// TwinCAT 3 PLC project MainProgram
// ProgramVersion: 3.1.4023.0
// libraries:
//   Tc2_Standard, * (Beckhoff Automation GmbH)
//   Tc2_System, * (Beckhoff Automation GmbH)
//   Tc3_Module, * (Beckhoff Automation GmbH)
// project tree:
//   DUT/ POS_Control.TcDUT, POS_Control_Control.TcDUT, POS_Status.TcDUT, POS_Status_Status.TcDUT, STM_Control.TcDUT, STM_Control_Control.TcDUT, STM_Status.TcDUT, STM_Status_Status.TcDUT, ST_PosInterface.TcDUT
//   GVLs/ GVL_IO.TcGVL
//   / PlcTask.TcTTO
//   POUs/ MAIN.TcPOU, POU_Example2PositionalMoves.TcPOU, POU_ExampleDynamicMoves.TcPOU
// real-time tasks:
//   TASK PlcTask: cycle T#10ms, priority 20, ADS port 350
//   TASK VnTask ImgAcq (FileSource1): cycle T#10ms, priority 5, ADS port 351
// I/O:
//   DEVICE Device 1 (Beckhoff CCAT)
//   DEVICE Device 2 (EtherCAT), AmsNetId 5.68.118.43.3.1
//     Term 1 (EK1200) [EK1200-5000 EtherCAT Power supply (2A E-Bus)]
//       Term 2 (EL7031) [EL7031 1Ch. Stepper motor output stage (24V, 1.5A)]
//       Term 3 (EL9011) [EL9011 End Terminal]
// variable links:
//   MainProgram Instance <-> Device 2 (EtherCAT)/Term 1 (EK1200)/Term 2 (EL7031)
//     PlcTask Inputs/GVL_IO.Axis.PosStatus/ActualDriveTime <-> POS Status/Actual drive time
//     PlcTask Inputs/GVL_IO.Axis.PosStatus/ActualPosition <-> POS Status/Actual position
//     PlcTask Inputs/GVL_IO.Axis.PosStatus/ActualVelocity <-> POS Status/Actual velocity
//     PlcTask Inputs/GVL_IO.Axis.PosStatus/Status <-> POS Status/Status
//     PlcTask Inputs/GVL_IO.Axis.StmStatus/Status <-> STM Status/Status
//     PlcTask Outputs/GVL_IO.Axis.PosControl/Acceleration <-> POS Control/Acceleration
//     PlcTask Outputs/GVL_IO.Axis.PosControl/Control <-> POS Control/Control
//     PlcTask Outputs/GVL_IO.Axis.PosControl/Deceleration <-> POS Control/Deceleration
//     PlcTask Outputs/GVL_IO.Axis.PosControl/StartType <-> POS Control/Start type
//     PlcTask Outputs/GVL_IO.Axis.PosControl/TargetPosition <-> POS Control/Target position
//     PlcTask Outputs/GVL_IO.Axis.PosControl/Velocity <-> POS Control/Velocity
//     PlcTask Outputs/GVL_IO.Axis.StmControl/Control <-> STM Control/Control

CONFIGURATION MainProgram
    RESOURCE PLC ON TwinCAT3
        TASK PlcTask(INTERVAL := T#10ms, PRIORITY := 20);
        PROGRAM MAIN WITH PlcTask : MAIN;
    END_RESOURCE
END_CONFIGURATION

// ---- DUT/POS_Control.TcDUT
TYPE POS_Control :
STRUCT
	Control : POS_Control_Control;
	TargetPosition : UDINT;
	Velocity : INT;
	StartType : UINT;
	Acceleration : UINT;
	Deceleration : UINT;
END_STRUCT
END_TYPE

// ---- DUT/POS_Control_Control.TcDUT
TYPE POS_Control_Control :
STRUCT
	Execute : BIT;
	EmergencyStop : BIT;
	
	{attribute 'hide'}
	padding_0_2	: BIT;
	{attribute 'hide'}
	padding_0_3	: BIT;
	{attribute 'hide'}
	padding_0_4	: BIT;
	{attribute 'hide'}
	padding_0_5	: BIT;
	{attribute 'hide'}
	padding_0_6	: BIT;
	{attribute 'hide'}
	padding_0_7	: BIT;
	{attribute 'hide'}
	padding_1_0	: BIT;
	{attribute 'hide'}
	padding_1_1	: BIT;
	{attribute 'hide'}
	padding_1_2	: BIT;
	{attribute 'hide'}
	padding_1_3	: BIT;
	{attribute 'hide'}
	padding_1_4	: BIT;
	{attribute 'hide'}
	padding_1_5	: BIT;
	{attribute 'hide'}
	padding_1_6	: BIT;
	{attribute 'hide'}
	padding_1_7	: BIT;
END_STRUCT
END_TYPE

// ---- DUT/POS_Status.TcDUT
TYPE POS_Status :
STRUCT
	Status : POS_Status_Status;
	ActualPosition : UDINT;
	ActualVelocity : INT;
	ActualDriveTime : UDINT;
END_STRUCT
END_TYPE

// ---- DUT/POS_Status_Status.TcDUT
TYPE POS_Status_Status :
STRUCT
	Busy : BIT;
	InTarget : BIT;
	Warning : BIT;
	Error : BIT;
	Calibrated : BIT;
	Accelerate : BIT;
	Decelerate : BIT;
	
	{attribute 'hide'}
	padding_0_7	: BIT;
	{attribute 'hide'}
	padding_1_0	: BIT;
	{attribute 'hide'}
	padding_1_1	: BIT;
	{attribute 'hide'}
	padding_1_2	: BIT;
	{attribute 'hide'}
	padding_1_3	: BIT;
	{attribute 'hide'}
	padding_1_4	: BIT;
	{attribute 'hide'}
	padding_1_5	: BIT;
	{attribute 'hide'}
	padding_1_6	: BIT;
	{attribute 'hide'}
	padding_1_7	: BIT;
END_STRUCT
END_TYPE

// ---- DUT/STM_Control.TcDUT
TYPE STM_Control :
STRUCT
	Control : STM_Control_Control;
END_STRUCT
END_TYPE

// ---- DUT/STM_Control_Control.TcDUT
TYPE STM_Control_Control :
STRUCT
	Enable : BIT;
	Reset : BIT;
	ReduceTorque : BIT;
	
	{attribute 'hide'}
	padding_0_3	: BIT;
	{attribute 'hide'}
	padding_0_4	: BIT;
	{attribute 'hide'}
	padding_0_5	: BIT;
	{attribute 'hide'}
	padding_0_6	: BIT;
	{attribute 'hide'}
	padding_0_7	: BIT;
	{attribute 'hide'}
	padding_1_0	: BIT;
	{attribute 'hide'}
	padding_1_1	: BIT;
	{attribute 'hide'}
	padding_1_2	: BIT;
	{attribute 'hide'}
	padding_1_3	: BIT;
	{attribute 'hide'}
	padding_1_4	: BIT;
	{attribute 'hide'}
	padding_1_5	: BIT;	
	{attribute 'hide'}
	padding_1_6	: BIT;
	{attribute 'hide'}
	padding_1_7	: BIT;
END_STRUCT
END_TYPE

// ---- DUT/STM_Status.TcDUT
TYPE STM_Status :
STRUCT
	Status : STM_Status_Status;
END_STRUCT
END_TYPE

// ---- DUT/STM_Status_Status.TcDUT
TYPE STM_Status_Status :
STRUCT
	ReadyToEnable : BIT;
	Ready : BIT;
	Warning : BIT;
	Error : BIT;
	MovingPositive : BIT;
	MovingNegative : BIT;
	TorqueReduced : BIT;
	
	{attribute 'hide'}
	padding_0_7	: BIT;
	{attribute 'hide'}
	padding_1_0	: BIT;
	{attribute 'hide'}
	padding_1_1	: BIT;
	{attribute 'hide'}
	padding_1_2	: BIT;
	
	DigitalInput1 : BIT;
	DigitalInput2 : BIT;
	SyncError : BIT;
	
	{attribute 'hide'}
	padding_1_6	: BIT;
	
	TxPDOToggle : BIT;
END_STRUCT
END_TYPE

// ---- DUT/ST_PosInterface.TcDUT
TYPE ST_PosInterface :
STRUCT
	PosControl AT%Q* : POS_Control;
	PosStatus AT%I* : POS_Status;
	StmControl AT%Q* : STM_Control;
	StmStatus AT%I* : STM_Status;
END_STRUCT
END_TYPE

// ---- GVLs/GVL_IO.TcGVL
VAR_GLOBAL
	Axis : ST_PosInterface;
END_VAR

// ---- POUs/MAIN.TcPOU
PROGRAM MAIN
VAR	
END_VAR
VAR CONSTANT
END_VAR

// Only enable one example at a time. 
//-----------------------------------

POU_Example2PositionalMoves();
//POU_ExampleDynamicMoves();

END_PROGRAM

// ---- POUs/POU_Example2PositionalMoves.TcPOU
PROGRAM POU_Example2PositionalMoves
VAR
	bCycleEnable : BOOL; // set true to start motion
	iState : INT := -40;	
END_VAR
VAR CONSTANT
	ABSOLUTE : UINT := 16#0001;
	SET_CALIBRATION : UINT := 16#6E00;
END_VAR

CASE iState OF
		
	-40: // check for card errors and reset.
		IF Axis.PosStatus.Status.Error THEN 
			Axis.StmControl.Control.Reset := TRUE;
		ELSE
			Axis.StmControl.Control.Reset := FALSE;
			iState := iState + 10;
		END_IF
		
	-30: // wait for card to be ready.
		IF Axis.StmStatus.Status.ReadyToEnable THEN 
			Axis.StmControl.Control.Enable := TRUE;
			iState := iState + 10;
		END_IF
		
	-20: // set card to manually calibrated.
		IF Axis.StmStatus.Status.Ready THEN 
			Axis.PosControl.StartType := SET_CALIBRATION;
			Axis.PosControl.Control.Execute := TRUE;
			iState := iState + 10;
		END_IF
		
	-10: // Check for calibrated flag then enable
		IF Axis.PosStatus.Status.Calibrated THEN 
			Axis.PosControl.Control.Execute := FALSE;
			iState := iState + 10;
		END_IF
		
	0: // Start operation
		IF bCycleEnable THEN
			iState := 10;
		END_IF
		
	10: // Set demand extend movement
		Axis.PosControl.Acceleration := 1000;
		Axis.PosControl.Deceleration := 1000;
		Axis.PosControl.StartType := ABSOLUTE;
		Axis.PosControl.Velocity := 500;
		Axis.PosControl.TargetPosition := 20000;
		Axis.PosControl.Control.Execute := TRUE;
		
		IF Axis.PosStatus.ActualPosition = Axis.PosControl.TargetPosition THEN
			Axis.PosControl.Control.Execute := FALSE;
			iState := 20;
		END_IF
		
	20: // wait
		IF NOT Axis.PosStatus.Status.Busy THEN
			iState := 30;
		END_IF
		
	30: // Set demand retract movement
		Axis.PosControl.Acceleration := 2000;
		Axis.PosControl.Deceleration := 2000;
		Axis.PosControl.StartType := ABSOLUTE;
		Axis.PosControl.Velocity := 1000;
		Axis.PosControl.TargetPosition := 0;
		Axis.PosControl.Control.Execute := TRUE;
		
		IF Axis.PosStatus.ActualPosition = Axis.PosControl.TargetPosition THEN
			Axis.PosControl.Control.Execute := FALSE;
			iState := 40;
		END_IF
		
	40: // wait
		IF NOT Axis.PosStatus.Status.Busy THEN
			iState := 0;
		END_IF
		
END_CASE

END_PROGRAM

// ---- POUs/POU_ExampleDynamicMoves.TcPOU
PROGRAM POU_ExampleDynamicMoves
VAR
	bCycleEnable : BOOL; // set true to start motion
	iState : INT := -40;	
END_VAR
VAR CONSTANT
	ABSOLUTE : UINT := 16#0001;
	ABSOLUTE_CHANGE : UINT := 16#1001;
	SET_CALIBRATION : UINT := 16#6E00;
END_VAR

CASE iState OF
		
	-40: // check for card errors and reset.
		IF Axis.PosStatus.Status.Error THEN 
			Axis.StmControl.Control.Reset := TRUE;
		ELSE
			Axis.StmControl.Control.Reset := FALSE;
			iState := iState + 10;
		END_IF
		
	-30: // wait for card to be ready.
		IF Axis.StmStatus.Status.ReadyToEnable THEN 
			Axis.StmControl.Control.Enable := TRUE;
			iState := iState + 10;
		END_IF
		
	-20: // set card to manually calibrated.
		IF Axis.StmStatus.Status.Ready THEN 
			Axis.PosControl.StartType := SET_CALIBRATION;
			Axis.PosControl.Control.Execute := TRUE;
			iState := iState + 10;
		END_IF
		
	-10: // Check for calibrated flag then enable
		IF Axis.PosStatus.Status.Calibrated THEN 
			Axis.PosControl.Control.Execute := FALSE;
			iState := iState + 10;
		END_IF
		
	0: // Start operation
		IF bCycleEnable AND NOT Axis.PosStatus.Status.Busy THEN 
			iState := iState + 10;
		END_IF
		
	10: // Set first move
		Axis.PosControl.Acceleration := 4000;
		Axis.PosControl.Deceleration := 4000;
		Axis.PosControl.StartType := ABSOLUTE;
		Axis.PosControl.Velocity := 4000;
		Axis.PosControl.TargetPosition := 80000;
		Axis.PosControl.Control.Execute := TRUE;

		IF Axis.PosStatus.ActualPosition > 1000 THEN
			iState := iState + 10;
		END_IF
		
	20: // dynamic change
	
		Axis.PosControl.StartType := ABSOLUTE_CHANGE;
		Axis.PosControl.TargetPosition := 40000;
		
		IF Axis.PosStatus.ActualPosition > 30000 THEN
			Axis.PosControl.StartType := ABSOLUTE;
			iState := iState + 10;
		END_IF

	30: // dynamic change
	
		Axis.PosControl.StartType := ABSOLUTE_CHANGE;
		Axis.PosControl.TargetPosition := 20000;
		
		IF Axis.PosStatus.ActualPosition < 25000 THEN
			Axis.PosControl.StartType := ABSOLUTE;
			iState := iState + 10;	
		END_IF
	
	40: // dynamic change
	
		Axis.PosControl.StartType := ABSOLUTE_CHANGE;
		Axis.PosControl.TargetPosition := 80000;
		
		IF Axis.PosStatus.ActualPosition > 61000 THEN
			Axis.PosControl.StartType := ABSOLUTE;
			iState := iState + 10;
		END_IF
		
	50: // dynamic change and end
	
		Axis.PosControl.StartType := ABSOLUTE_CHANGE;
		Axis.PosControl.TargetPosition := 0;
		
		IF Axis.PosStatus.ActualPosition = Axis.PosControl.TargetPosition THEN
			Axis.PosControl.Control.Execute := FALSE;
			iState := 0;
		END_IF
		
END_CASE

END_PROGRAM
